// TIA Portal V16 export
// export: Created 2021-07-12T14:47:20.0455708Z, ExportSetting WithDefaults, DisplayName Totally Integrated Automation Portal, DisplayVersion V16, DisplayName TIA Portal Version Control Interface, DisplayVersion V16, DisplayName TIA Portal Openness, DisplayVersion V16, DisplayName STEP 7 Professional, DisplayVersion V16, DisplayName STEP 7 Safety, DisplayVersion V16, DisplayName WinCC Professional, DisplayVersion V16
TYPE "LSimaHydTO_typeVCharMeasured"
TITLE = LSimaHydTO_typeVCharMeasured
// Measured Values in one direction
// stored: IsFailsafeCompliant false
   STRUCT
      qOutput : Array[0.."LSIMAHYD_VCHAR_POINTS_UPPER_LIMIT"] of Real;   // manipulated variable
      velocity : Array[0.."LSIMAHYD_VCHAR_POINTS_UPPER_LIMIT"] of Real;   // velocity
      maxVelocity : Real;   // max. measured velocity
      minQOutput : Real;   // min. manipulated variable
      maxQOutput : Real;   // max. manipulated variable
      maxIndexMeasurement : Int;   // measurement was made up to this index
      coarseBegin : Real;   // coarse area begins by this index
   END_STRUCT;
END_TYPE
